{attribute 'qualified_only'}
VAR_GLOBAL
	
	outJson : STRING(2000);

END_VAR
	
VAR_GLOBAL CONSTANT
	
	singleLiteralBool : STRING(1000) := '	
		{
		  "nodes": [
			{
			  "id": "1",
			  "type": "PLC Basic/Literals/BOOL",
			  "order": 0,
			  "mode": 0,
			  "outputs": [
				{ "name": "out", "type": "BOOL", "links": null }
			  ],
			  "title": "Literal_BOOL",
			  "properties": { "value": true }
			}
		  ],
		  "uuid": "20790db0-072c-4676-bf41-a34c1013bf75"
		}
	';
	
	literalBoolLinkedToDisplayBool : STRING(1000) := '
		{
		  "nodes": [
			{
			  "id": "2",
			  "type": "PLC Basic/Display/BOOL",
			  "order": 1,
			  "mode": 0,
			  "inputs": [
				{
				  "name": "in",
				  "type": "BOOL"
				}
			  ],
			  "title": "Display_BOOL"
			},
			{
			  "id": "1",
			  "type": "PLC Basic/Literals/BOOL",
			  "order": 0,
			  "mode": 0,
			  "outputs": [
				{
				  "name": "out",
				  "type": "BOOL"
				}
			  ],
			  "title": "Literal_BOOL",
			  "properties": {
				"value": true
			  }
			}
		  ],
		  "links": [
			[
			  "1",
			  "1",
			  "out",
			  "2",
			  "in"
			]
		  ],
		  "uuid": "8506b771-8bd4-4160-984e-e0e4aa529fec"
		}
	';
	
END_VAR

(* stored: Version 1.1.0.1, ProductVersion 3.1.4024.12
   GVL TestJson: Id {1cdc49ca-6866-01b4-0af3-ddaff08f436e} *)
